FUNCTION Camera_Set_Bool : Buffer_Error
VAR_INPUT
	Num : USINT;
	In : BOOL;
END_VAR

VAR_IN_OUT
	Camera : Cognex_Camera;
END_VAR

Camera_Set_Bool := Set_Bool_Fom_Buffer(	In:= In, 
										Num:= Num, 
										Layout:= Camera.Ouput_Buffer_Layout, 
										Buffer:= Camera.User_Data.UserData)

END_FUNCTION

(* stored: Version 1.1.0.1, ProductVersion 3.1.4024.10
   POU Camera_Set_Bool: Id {bf8a1094-fd99-4174-a00c-8e948d92e357}, SpecialFunc None *)
